// Mitsubishi GX Works2 project: 서보3   PLC: Q02/Q02H

PROGRAM MAIN
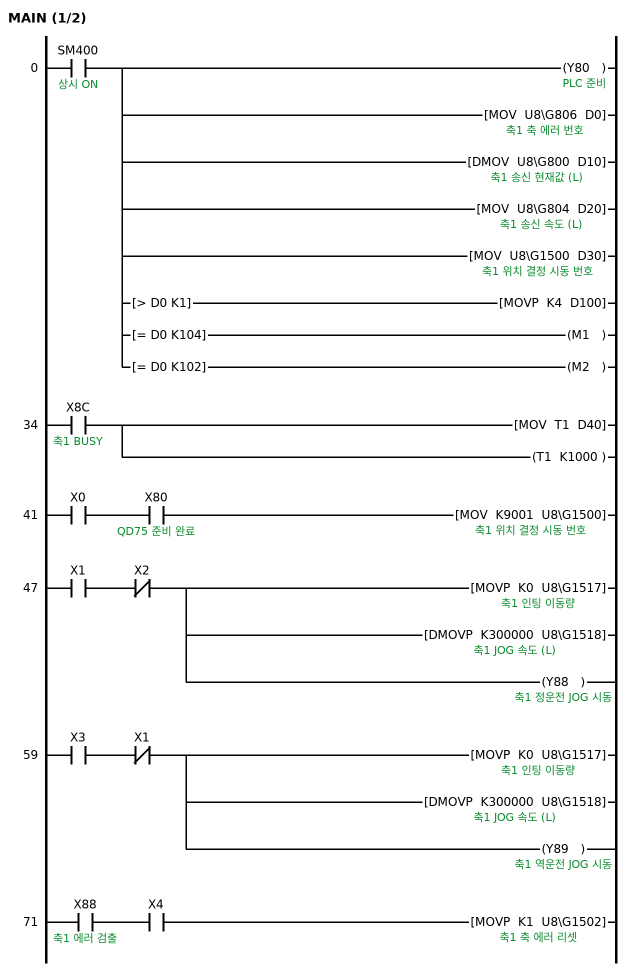
0     LD      SM400  ; 상시 ON
      OUT     Y80  ; PLC 준비
      MOV     U8\G806 D0  ; 축1 축 에러 번호
      DMOV    U8\G800 D10  ; 축1 송신 현재값 (L)
      MOV     U8\G804 D20  ; 축1 송신 속도 (L)
      MOV     U8\G1500 D30  ; 축1 위치 결정 시동 번호
      MPS
      AND>    D0 K1
      MOVP    K4 D100
      MRD
      AND=    D0 K104
      OUT     M1
      MPP
      AND=    D0 K102
      OUT     M2
34    LD      X8C  ; 축1 BUSY
      MOV     T1 D40
      OUT     T1 K1000
41    LD      X0
      AND     X80  ; QD75 준비 완료
      MOV     K9001 U8\G1500
47    LD      X1
      ANI     X2
      MOVP    K0 U8\G1517  ; 축1 인팅 이동량
      DMOVP   K300000 U8\G1518  ; 축1 JOG 속도 (L)
      OUT     Y88  ; 축1 정운전 JOG 시동
59    LD      X3
      ANI     X1
      MOVP    K0 U8\G1517
      DMOVP   K300000 U8\G1518
      OUT     Y89  ; 축1 역운전 JOG 시동
71    LD      X88  ; 축1 에러 검출
      AND     X4
      MOVP    K1 U8\G1502  ; 축1 축 에러 리셋
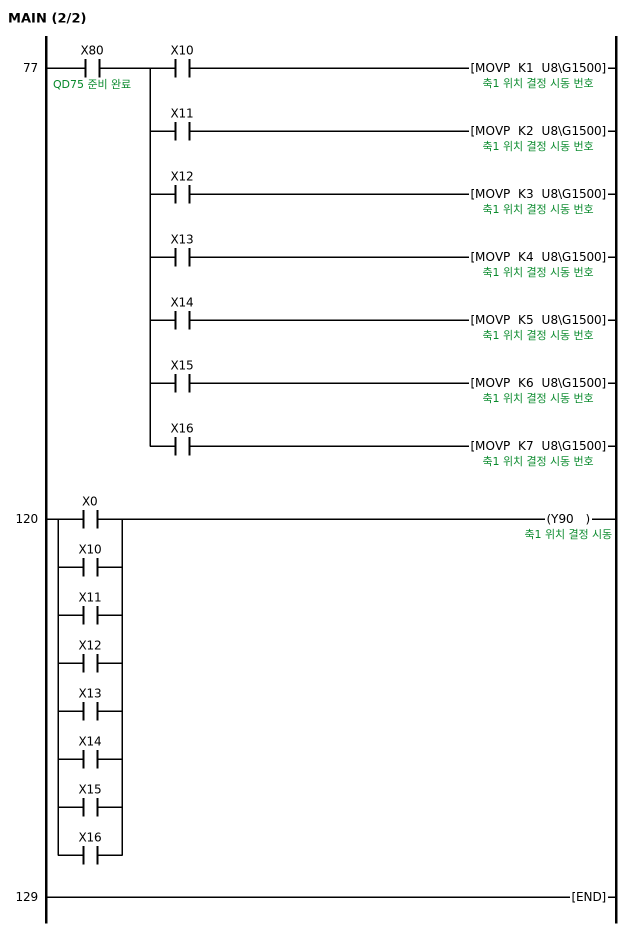
77    LD      X80  ; QD75 준비 완료
      MPS
      AND     X10
      MOVP    K1 U8\G1500
      MRD
      AND     X11
      MOVP    K2 U8\G1500
      MRD
      AND     X12
      MOVP    K3 U8\G1500
      MRD
      AND     X13
      MOVP    K4 U8\G1500
      MRD
      AND     X14
      MOVP    K5 U8\G1500
      MRD
      AND     X15
      MOVP    K6 U8\G1500
      MPP
      AND     X16
      MOVP    K7 U8\G1500
120   LD      X0
      OR      X10
      OR      X11
      OR      X12
      OR      X13
      OR      X14
      OR      X15
      OR      X16
      OUT     Y90  ; 축1 위치 결정 시동
129   END
END_PROGRAM

// device comments not shown above
X81  ; 동기용 플래그
X84  ; 축1 M 코드 ON
X85  ; 축2 M 코드 ON
X89  ; 축2 에러 검출
X8D  ; 축2 BUSY
X90  ; 축1 시동 완료
X91  ; 축2 시동 완료
X94  ; 축1 위치 결정 완료
X95  ; 축2 위치 결정 완료
Y84  ; 축1 축 정지
Y85  ; 축2 축 정지
Y8A  ; 축2 정운전 JOG 시동
Y8B  ; 축2 역운전 JOG 시동
Y91  ; 축2 위치 결정 시동
Y94  ; 축1 실행 금지 플래그
Y95  ; 축2 실행 금지 플래그
